// Mitsubishi GX Works2 project: n07   PLC: Q02/Q02H

PROGRAM MAIN
VAR
  CTU_1 : CTU;
  CTU_2 : CTU;
  CTD_1 : CTD;
END_VAR
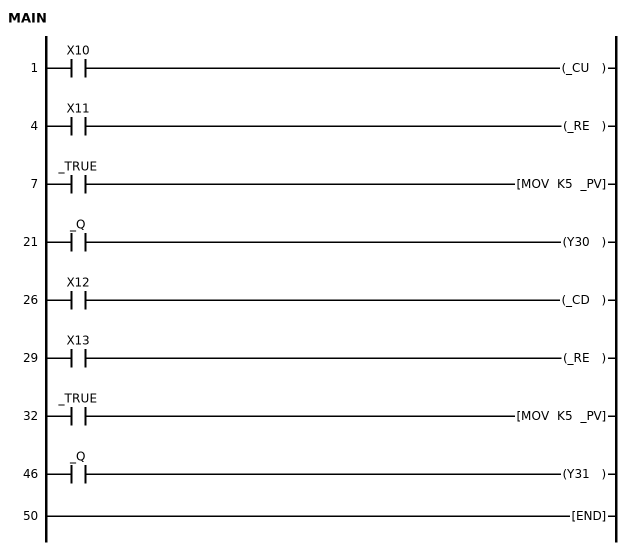
; FB BLK START CTU(CTU_2)
1     LD      X10
      OUT     _CU
4     LD      X11
      OUT     _RE
7     LD      _TRUE
      MOV     K5 _PV
; FB START
; FB_NAME CTU
; INSTANCE_NAME CTU_2
; FB IN_B:CU
; FB OUT_Q:B
; FB IN_B:RE
; FB OUT_CV:W
; FB IN_W:PV
; FB END
21    LD      _Q
      OUT     Y30
; FB BLK END
; FB BLK START CTD(CTD_1)
26    LD      X12
      OUT     _CD
29    LD      X13
      OUT     _RE
32    LD      _TRUE
      MOV     K5 _PV
; FB START
; FB_NAME CTD
; INSTANCE_NAME CTD_1
; FB IN_B:CD
; FB OUT_Q:B
; FB IN_B:RE
; FB OUT_CV:W
; FB IN_W:PV
; FB END
46    LD      _Q
      OUT     Y31
; FB BLK END
50    END
END_PROGRAM

FUNCTION_BLOCK CTU
VAR_INPUT
  CU : BOOL;
  RE : BOOL;
  PV : INT;
END_VAR
VAR_OUTPUT
  Q : BOOL;
  CV : INT;
END_VAR
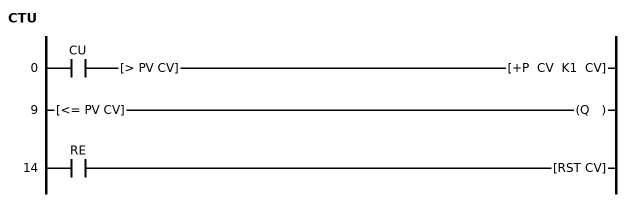
0     LD      CU
      AND>    PV CV
      +P      CV K1 CV
9     LD<=    PV CV
      OUT     Q
14    LD      RE
      RST     CV
END_FUNCTION_BLOCK

FUNCTION_BLOCK CTD
VAR_INPUT
  RE : BOOL;
  CD : BOOL;
END_VAR
VAR_OUTPUT
  Q : BOOL;
  CV : INT;
END_VAR
VAR_INPUT
  PV : INT;
END_VAR
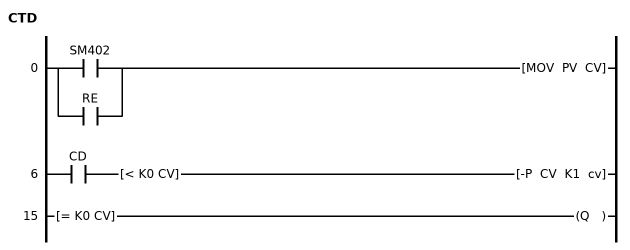
0     LD      SM402
      OR      RE
      MOV     PV CV
6     LD      CD
      AND<    K0 CV
      -P      CV K1 cv
15    LD=     K0 CV
      OUT     Q
END_FUNCTION_BLOCK
